(* Logix 5000 project; controller cal1615 1756-L62 rev 16.20; software revision 16.05; part 63 of 78 *)
(* tags used below, declared in another part *)
   FAULT : BOOL;   // Fault AFI
   HMI : BOOL;   // AFI HMI
   p01_recipe_active : recipe;   // Active Recipe
   p01r09_pb_global_reset : BOOL;   // System Modes PB: Global Fault Reset
   p26_ao_dia_a : REAL;   // Upper Poly Letoff Analog Input Letoff A Diameter
   p26_ao_dia_b : REAL;   // Upper Poly Letoff Analog Input Letoff B Diameter
   p26_dint_to_hmi : DINT[16];   // Upper Poly Letoff Dint to HMI
   p26_inactive_tension_sp : REAL;
   p26r01 : routine;   // Upper Poly Letoff
   p26r03_upper_A_tension_on : BOOL;
   p26r03_upper_B_tension_on : BOOL;
   p26r08 : routine;   // Upper Poly Letoff Warnings
   p26r08_timer_fault : TIMER[4];   // Upper Poly Letoff Warnings Fault Delay
   p26r08_timer_warning : TIMER[4];   // Upper Poly Letoff Warnings Warning Delay
   p26r09 : routine;   // Upper Poly Letoff Modes
   p26r09_timer_fault : TIMER[4];   // Lower Poly Letoff Modes Fault Delay
   p26r09_timer_warning : TIMER[4];   // Lower Poly Letoff Modes Warning Delay
   p26r10 : routine;   // Upper Poly Letoff Tension
   p26r10_timer_fault : TIMER[4];   // Lower Poly Letoff Fault Delay
   p26r10_timer_warning : TIMER[4];   // Lower Poly Letoff Warning Delay
   p26r10_ula_selected_tension : REAL;   // Upper Poly Letoff Tension A Selected Tension
   p26r10_ulb_selected_tension : REAL;   // Upper Poly Letoff Tension B Selected Tension
   p26r10_unwind_a_brake_torque : REAL;   // Upper Poly Letoff Tension Letoff A Brake Torque
   p26r10_unwind_a_dia_ft : REAL;   // Upper Poly Letoff Tension Diameter A [ft]
   p26r10_unwind_b_brake_torque : REAL;   // Upper Poly Letoff Tension Letoff B Brake Torque
   p26r10_unwind_b_dia_ft : REAL;   // Upper Poly Letoff Tension Diameter B [ft]
   p27r01 : routine;   // Winder Main
(* P26_Upper_Poly_Letoff, continued *)

ROUTINE R08_Warnings   (* ladder *)
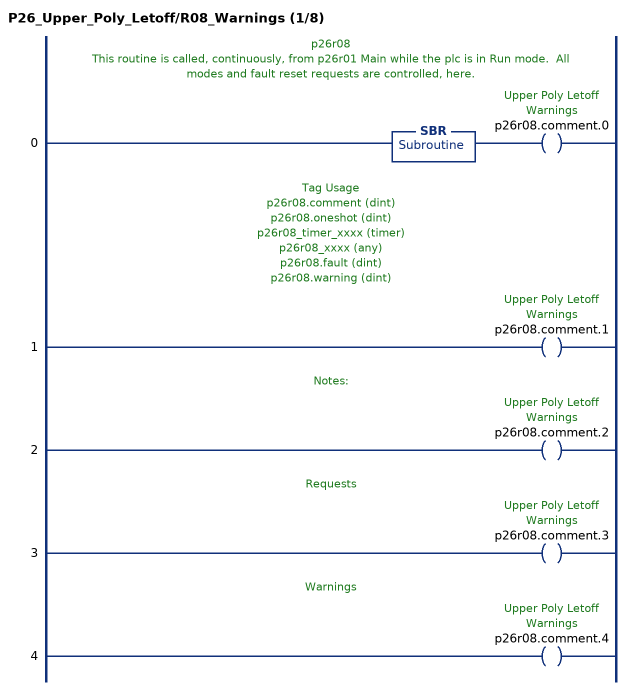
   // p26r08
   // This routine is called, continuously, from p26r01 Main while the plc is in Run mode.  All modes and fault reset requests are controlled, here.
   0: SBR()OTE(p26r08.comment.0);
   // Tag Usage
   // p26r08.comment (dint)
   // p26r08.oneshot (dint)
   // p26r08_timer_xxxx (timer)
   // p26r08_xxxx (any)
   // p26r08.fault (dint)
   // p26r08.warning (dint)
   1: OTE(p26r08.comment.1);
   // Notes:
   2: OTE(p26r08.comment.2);
   // Requests
   3: OTE(p26r08.comment.3);
   // Warnings
   4: OTE(p26r08.comment.4);
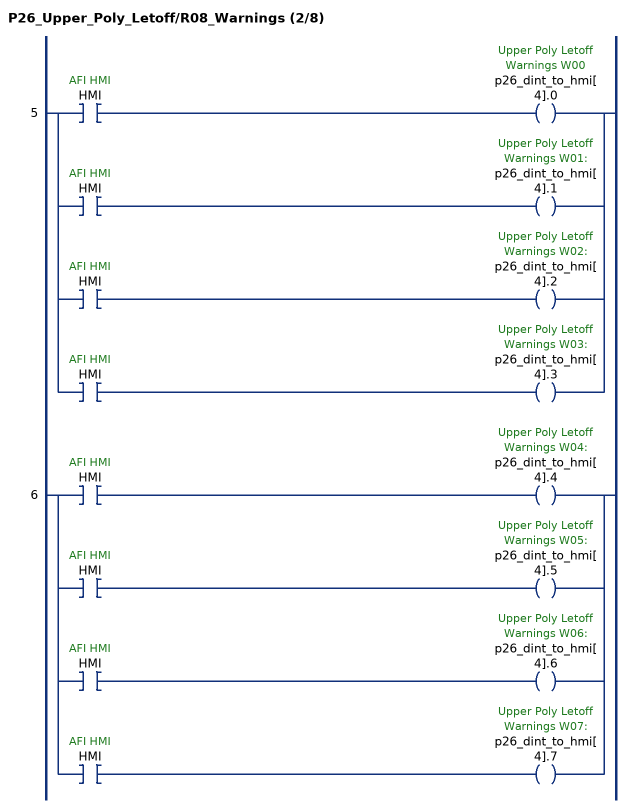
   5: [XIC(HMI) OTE(p26_dint_to_hmi[4].0) ,XIC(HMI) OTE(p26_dint_to_hmi[4].1) ,XIC(HMI) OTE(p26_dint_to_hmi[4].2) ,XIC(HMI) OTE(p26_dint_to_hmi[4].3) ];
   6: [XIC(HMI) OTE(p26_dint_to_hmi[4].4) ,XIC(HMI) OTE(p26_dint_to_hmi[4].5) ,XIC(HMI) OTE(p26_dint_to_hmi[4].6) ,XIC(HMI) OTE(p26_dint_to_hmi[4].7) ];
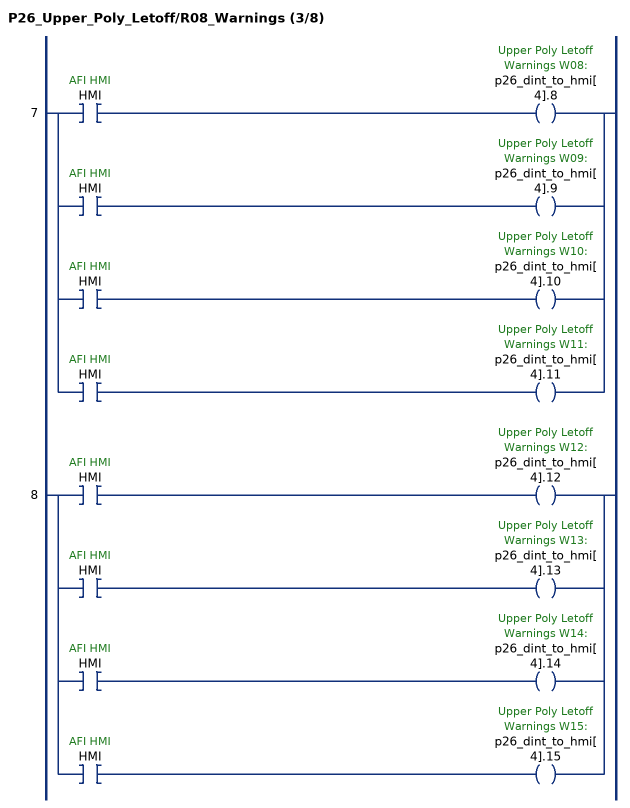
   7: [XIC(HMI) OTE(p26_dint_to_hmi[4].8) ,XIC(HMI) OTE(p26_dint_to_hmi[4].9) ,XIC(HMI) OTE(p26_dint_to_hmi[4].10) ,XIC(HMI) OTE(p26_dint_to_hmi[4].11) ];
   8: [XIC(HMI) OTE(p26_dint_to_hmi[4].12) ,XIC(HMI) OTE(p26_dint_to_hmi[4].13) ,XIC(HMI) OTE(p26_dint_to_hmi[4].14) ,XIC(HMI) OTE(p26_dint_to_hmi[4].15) ];
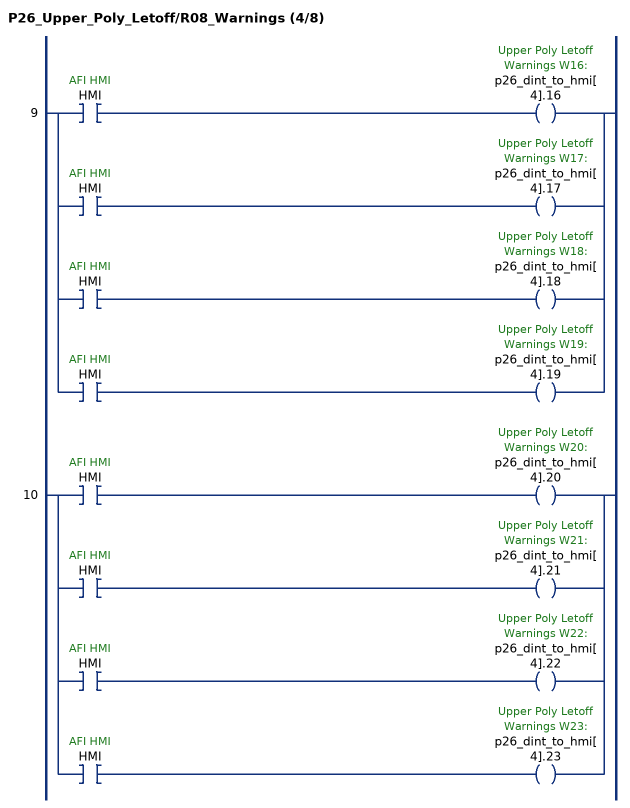
   9: [XIC(HMI) OTE(p26_dint_to_hmi[4].16) ,XIC(HMI) OTE(p26_dint_to_hmi[4].17) ,XIC(HMI) OTE(p26_dint_to_hmi[4].18) ,XIC(HMI) OTE(p26_dint_to_hmi[4].19) ];
   10: [XIC(HMI) OTE(p26_dint_to_hmi[4].20) ,XIC(HMI) OTE(p26_dint_to_hmi[4].21) ,XIC(HMI) OTE(p26_dint_to_hmi[4].22) ,XIC(HMI) OTE(p26_dint_to_hmi[4].23) ];
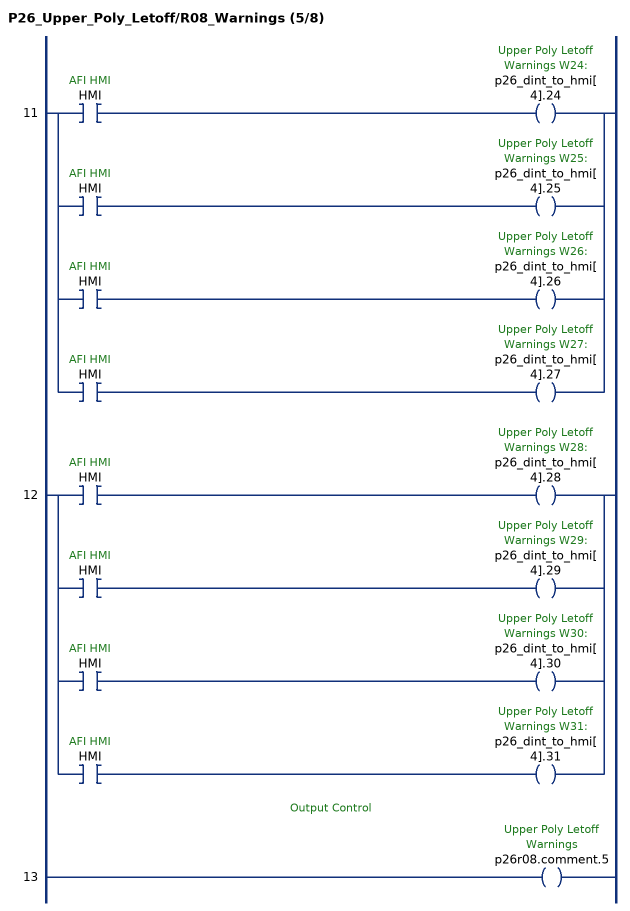
   11: [XIC(HMI) OTE(p26_dint_to_hmi[4].24) ,XIC(HMI) OTE(p26_dint_to_hmi[4].25) ,XIC(HMI) OTE(p26_dint_to_hmi[4].26) ,XIC(HMI) OTE(p26_dint_to_hmi[4].27) ];
   12: [XIC(HMI) OTE(p26_dint_to_hmi[4].28) ,XIC(HMI) OTE(p26_dint_to_hmi[4].29) ,XIC(HMI) OTE(p26_dint_to_hmi[4].30) ,XIC(HMI) OTE(p26_dint_to_hmi[4].31) ];
   // Output Control
   13: OTE(p26r08.comment.5);
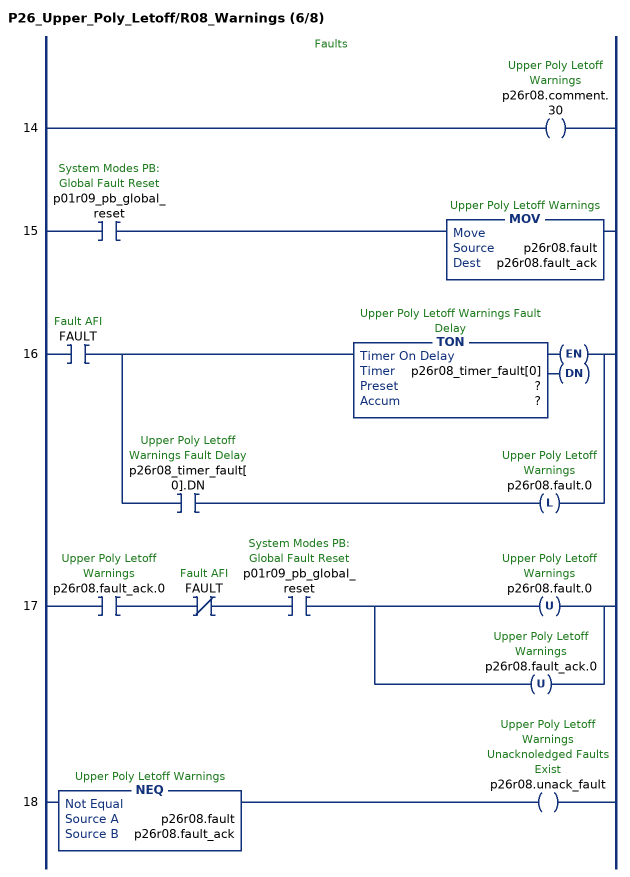
   // Faults
   14: OTE(p26r08.comment.30);
   15: XIC(p01r09_pb_global_reset)MOV(p26r08.fault,p26r08.fault_ack);
   16: XIC(FAULT)[TON(p26r08_timer_fault[0],?,?) ,XIC(p26r08_timer_fault[0].DN) OTL(p26r08.fault.0) ];
   17: XIC(p26r08.fault_ack.0)XIO(FAULT)XIC(p01r09_pb_global_reset)[OTU(p26r08.fault.0) ,OTU(p26r08.fault_ack.0) ];
   18: NEQ(p26r08.fault,p26r08.fault_ack)OTE(p26r08.unack_fault);
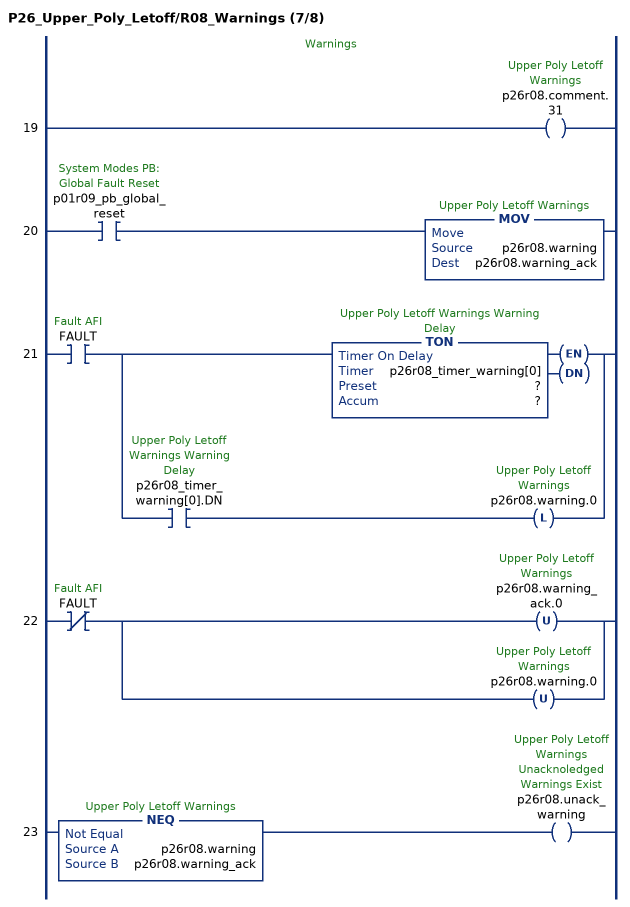
   // Warnings
   19: OTE(p26r08.comment.31);
   20: XIC(p01r09_pb_global_reset)MOV(p26r08.warning,p26r08.warning_ack);
   21: XIC(FAULT)[TON(p26r08_timer_warning[0],?,?) ,XIC(p26r08_timer_warning[0].DN) OTL(p26r08.warning.0) ];
   22: XIO(FAULT)[OTU(p26r08.warning_ack.0) ,OTU(p26r08.warning.0) ];
   23: NEQ(p26r08.warning,p26r08.warning_ack)OTE(p26r08.unack_warning);
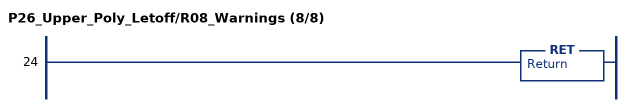
   24: RET();
END_ROUTINE

ROUTINE R09_Modes   (* ladder *)
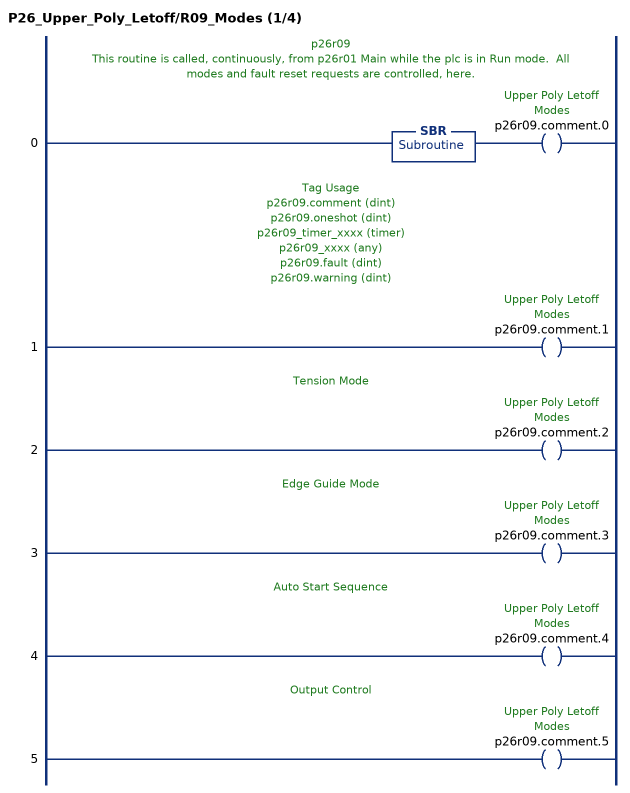
   // p26r09
   // This routine is called, continuously, from p26r01 Main while the plc is in Run mode.  All modes and fault reset requests are controlled, here.
   0: SBR()OTE(p26r09.comment.0);
   // Tag Usage
   // p26r09.comment (dint)
   // p26r09.oneshot (dint)
   // p26r09_timer_xxxx (timer)
   // p26r09_xxxx (any)
   // p26r09.fault (dint)
   // p26r09.warning (dint)
   1: OTE(p26r09.comment.1);
   // Tension Mode
   2: OTE(p26r09.comment.2);
   // Edge Guide Mode
   3: OTE(p26r09.comment.3);
   // Auto Start Sequence
   4: OTE(p26r09.comment.4);
   // Output Control
   5: OTE(p26r09.comment.5);
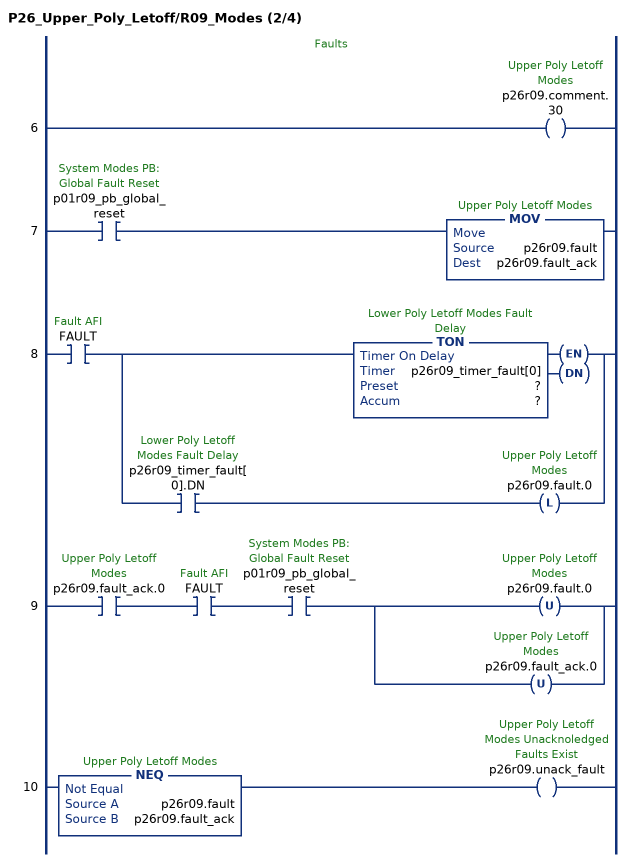
   // Faults
   6: OTE(p26r09.comment.30);
   7: XIC(p01r09_pb_global_reset)MOV(p26r09.fault,p26r09.fault_ack);
   8: XIC(FAULT)[TON(p26r09_timer_fault[0],?,?) ,XIC(p26r09_timer_fault[0].DN) OTL(p26r09.fault.0) ];
   9: XIC(p26r09.fault_ack.0)XIC(FAULT)XIC(p01r09_pb_global_reset)[OTU(p26r09.fault.0) ,OTU(p26r09.fault_ack.0) ];
   10: NEQ(p26r09.fault,p26r09.fault_ack)OTE(p26r09.unack_fault);
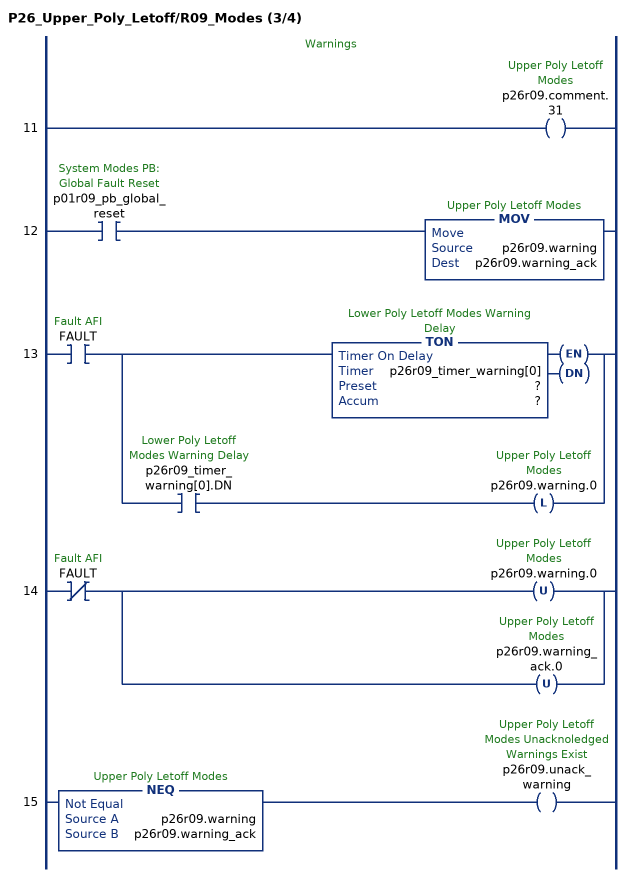
   // Warnings
   11: OTE(p26r09.comment.31);
   12: XIC(p01r09_pb_global_reset)MOV(p26r09.warning,p26r09.warning_ack);
   13: XIC(FAULT)[TON(p26r09_timer_warning[0],?,?) ,XIC(p26r09_timer_warning[0].DN) OTL(p26r09.warning.0) ];
   14: XIO(FAULT)[OTU(p26r09.warning.0) ,OTU(p26r09.warning_ack.0) ];
   15: NEQ(p26r09.warning,p26r09.warning_ack)OTE(p26r09.unack_warning);
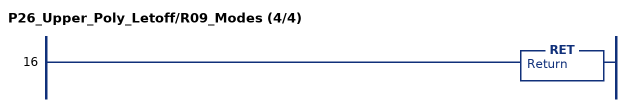
   16: RET();
END_ROUTINE

ROUTINE R10_Tension_A   (* ladder *)
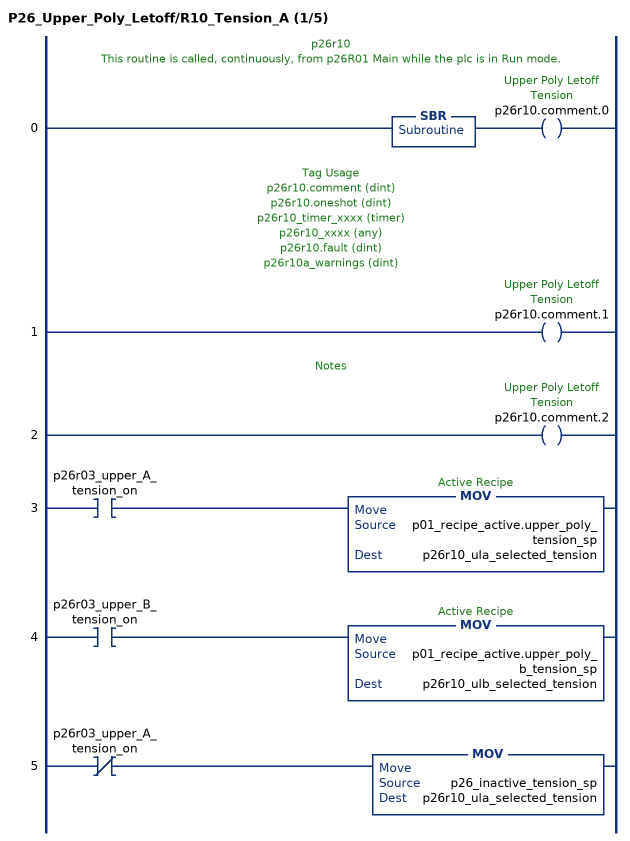
   // p26r10
   // This routine is called, continuously, from p26R01 Main while the plc is in Run mode.
   0: SBR()OTE(p26r10.comment.0);
   // Tag Usage
   // p26r10.comment (dint)
   // p26r10.oneshot (dint)
   // p26r10_timer_xxxx (timer)
   // p26r10_xxxx (any)
   // p26r10.fault (dint)
   // p26r10a_warnings (dint)
   1: OTE(p26r10.comment.1);
   // Notes
   2: OTE(p26r10.comment.2);
   3: XIC(p26r03_upper_A_tension_on)MOV(p01_recipe_active.upper_poly_tension_sp,p26r10_ula_selected_tension);
   4: XIC(p26r03_upper_B_tension_on)MOV(p01_recipe_active.upper_poly_b_tension_sp,p26r10_ulb_selected_tension);
   5: XIO(p26r03_upper_A_tension_on)MOV(p26_inactive_tension_sp,p26r10_ula_selected_tension);
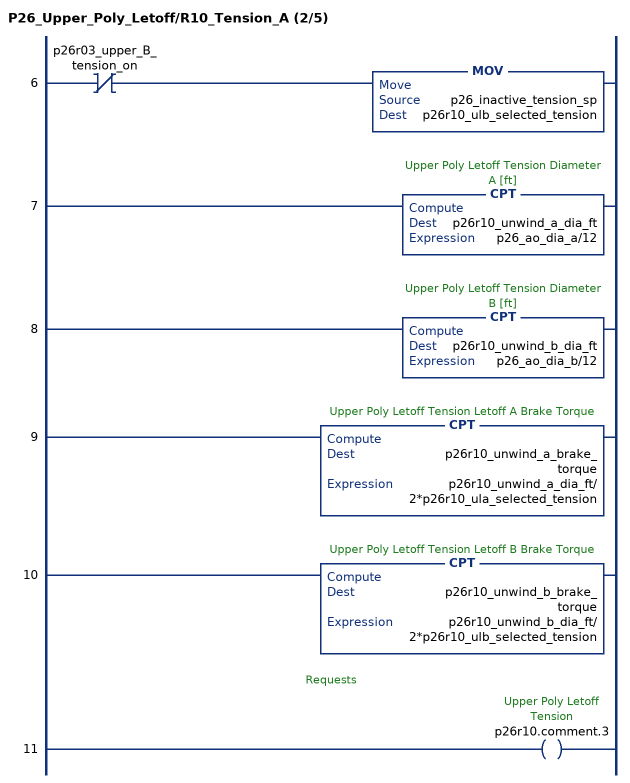
   6: XIO(p26r03_upper_B_tension_on)MOV(p26_inactive_tension_sp,p26r10_ulb_selected_tension);
   7: CPT(p26r10_unwind_a_dia_ft,p26_ao_dia_a/12);
   8: CPT(p26r10_unwind_b_dia_ft,p26_ao_dia_b/12);
   9: CPT(p26r10_unwind_a_brake_torque,p26r10_unwind_a_dia_ft/2*p26r10_ula_selected_tension);
   10: CPT(p26r10_unwind_b_brake_torque,p26r10_unwind_b_dia_ft/2*p26r10_ulb_selected_tension);
   // Requests
   11: OTE(p26r10.comment.3);
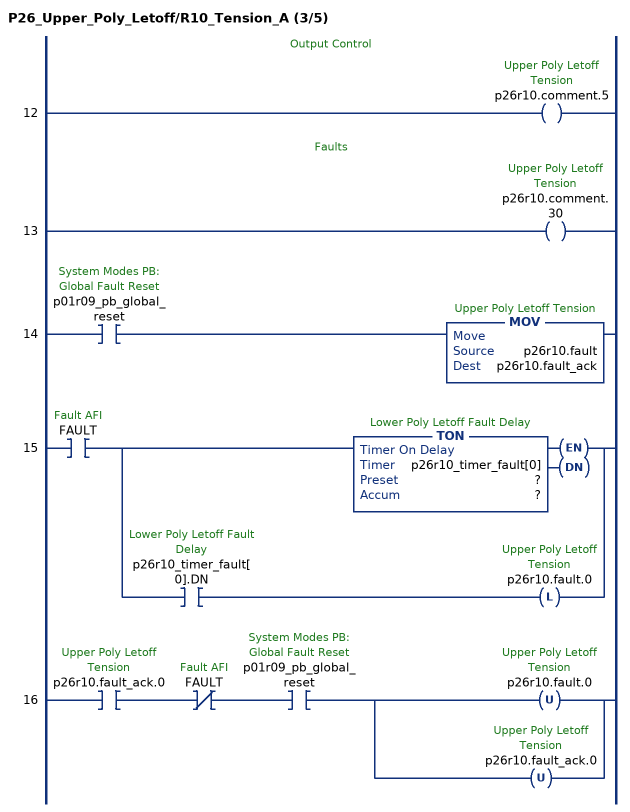
   // Output Control
   12: OTE(p26r10.comment.5);
   // Faults
   13: OTE(p26r10.comment.30);
   14: XIC(p01r09_pb_global_reset)MOV(p26r10.fault,p26r10.fault_ack);
   15: XIC(FAULT)[TON(p26r10_timer_fault[0],?,?) ,XIC(p26r10_timer_fault[0].DN) OTL(p26r10.fault.0) ];
   16: XIC(p26r10.fault_ack.0)XIO(FAULT)XIC(p01r09_pb_global_reset)[OTU(p26r10.fault.0) ,OTU(p26r10.fault_ack.0) ];
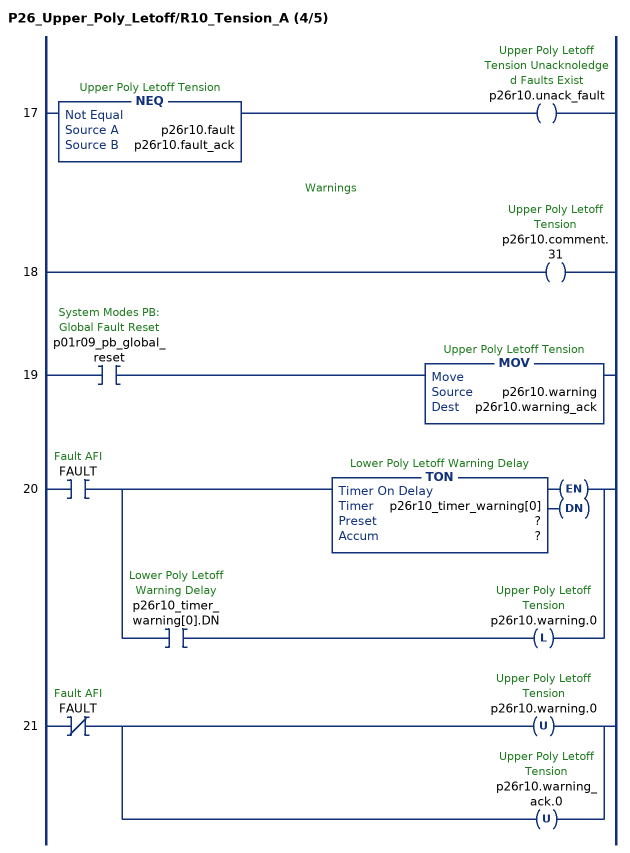
   17: NEQ(p26r10.fault,p26r10.fault_ack)OTE(p26r10.unack_fault);
   // Warnings
   18: OTE(p26r10.comment.31);
   19: XIC(p01r09_pb_global_reset)MOV(p26r10.warning,p26r10.warning_ack);
   20: XIC(FAULT)[TON(p26r10_timer_warning[0],?,?) ,XIC(p26r10_timer_warning[0].DN) OTL(p26r10.warning.0) ];
   21: XIO(FAULT)[OTU(p26r10.warning.0) ,OTU(p26r10.warning_ack.0) ];
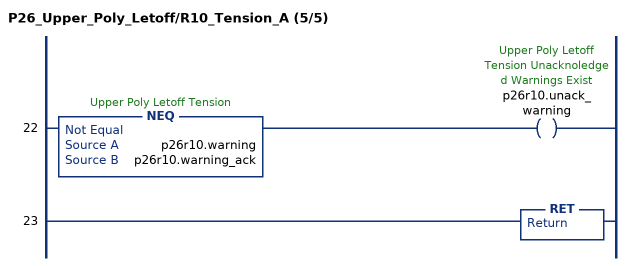
   22: NEQ(p26r10.warning,p26r10.warning_ack)OTE(p26r10.unack_warning);
   23: RET();
END_ROUTINE
END_PROGRAM

PROGRAM P27_Lower_Poly_Letoff   (* main routine R01_Main *)

ROUTINE R01_Main   (* ladder *)
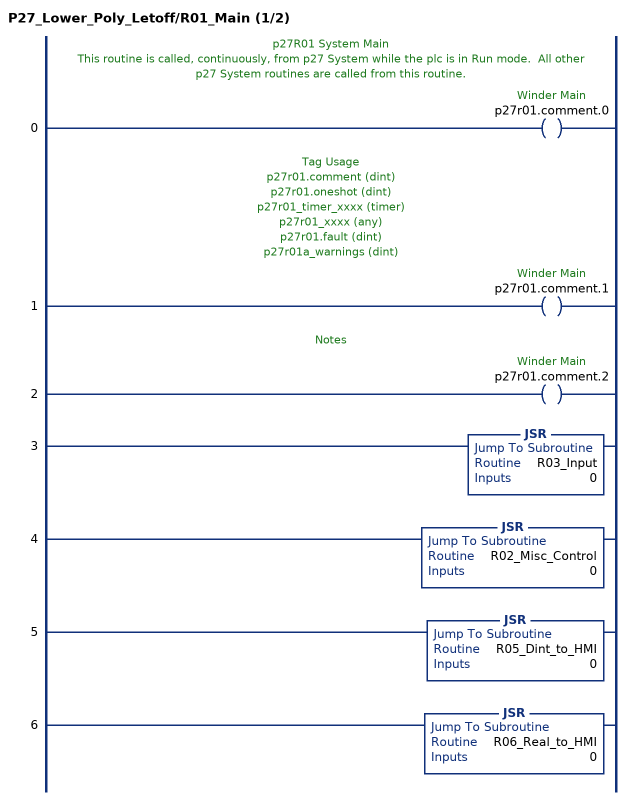
   // p27R01 System Main
   // This routine is called, continuously, from p27 System while the plc is in Run mode.  All other p27 System routines are called from this routine.
   0: OTE(p27r01.comment.0);
   // Tag Usage
   // p27r01.comment (dint)
   // p27r01.oneshot (dint)
   // p27r01_timer_xxxx (timer)
   // p27r01_xxxx (any)
   // p27r01.fault (dint)
   // p27r01a_warnings (dint)
   1: OTE(p27r01.comment.1);
   // Notes
   2: OTE(p27r01.comment.2);
   3: JSR(R03_Input,0);
   4: JSR(R02_Misc_Control,0);
   5: JSR(R05_Dint_to_HMI,0);
   6: JSR(R06_Real_to_HMI,0);
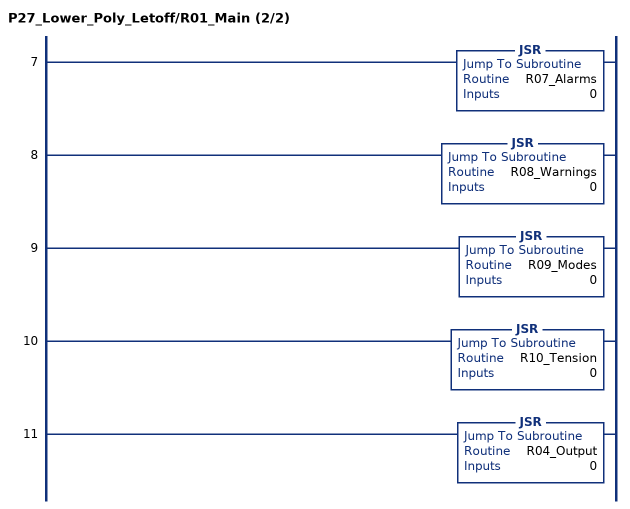
   7: JSR(R07_Alarms,0);
   8: JSR(R08_Warnings,0);
   9: JSR(R09_Modes,0);
   10: JSR(R10_Tension,0);
   11: JSR(R04_Output,0);
END_ROUTINE
